PROGRAM MAIN
VAR
	bRunOnlyOnce : BOOL := FALSE;
END_VAR

IF NOT bRunOnlyOnce THEN
	
	ADSLOGSTR(msgCtrlMask := ADSLOG_MSGTYPE_ERROR OR ADSLOG_MSGTYPE_LOG,
				msgFmtStr:= 'Hello World',
				strArg := '');
	bRunOnlyOnce := TRUE;
END_IF

END_PROGRAM

(* stored: Version 1.1.0.1, ProductVersion 3.1.4024.12
   POU MAIN: Id {6fa3cec0-cc11-4b91-8483-ce1d4f50e090}, SpecialFunc None *)
